TYPE Union_REAL :
UNION
	value : REAL;
	Packed : ARRAY[0..3] OF BYTE;
END_UNION
END_TYPE

(* stored: Version 1.1.0.1, ProductVersion 3.1.4024.13
   DUT Union_REAL: Id {4a15a7ff-499f-497c-acdf-6a173c7a94fb} *)
